INTERFACE I_DigitalCommandable

METHOD SetOn : E_RpcMethodResponse
VAR_INPUT
    eRequester : E_Requester := E_Requester.PROG;
END_VAR
END_METHOD

METHOD SetOff : E_RpcMethodResponse
VAR_INPUT
    eRequester : E_Requester := E_Requester.PROG;
END_VAR
END_METHOD

END_INTERFACE

(* stored: Version 1.1.0.1, ProductVersion 3.1.4026.12
   Itf I_DigitalCommandable: Id {c0000004-0000-0000-0000-000000000001}
   Method SetOn: Id {c0000004-0000-0000-1000-000000000001}
   Method SetOff: Id {c0000004-0000-0000-1000-000000000002} *)
